TYPE TcoUrRobotics_T2O_IntRegs_IO :
STRUCT
    bArray AT %I* : ARRAY[0..95] OF BYTE;
END_STRUCT
END_TYPE

(* stored: Version 1.1.0.1, ProductVersion 3.1.4024.12
   DUT TcoUrRobotics_T2O_IntRegs_IO: Id {fa563f9f-f364-07c1-17ca-b1b4df96b26d} *)
